FUNCTION F_NormSqQuat : LREAL
VAR_INPUT
    iQuat : I_Quat;
END_VAR


F_NormSqQuat := iQuat.w*iQuat.w + F_NormSqVec3(iQuat);

END_FUNCTION

(* stored: Version 1.1.0.1
   POU F_NormSqQuat: Id {42312887-5f96-4969-87c2-7747d5e51a97}, SpecialFunc None *)
